FUNCTION_BLOCK T_Cylinder IMPLEMENTS I_Cylinder
VAR_INPUT
END_VAR
VAR_OUTPUT
END_VAR
VAR
	output AT %Q* : BOOL;
END_VAR

METHOD PUBLIC Extend
VAR_INPUT
END_VAR
output := true;
END_METHOD

METHOD PUBLIC Retract
VAR_INPUT
END_VAR
output := false;
END_METHOD

END_FUNCTION_BLOCK

(* stored: Version 1.1.0.1, ProductVersion 3.1.4024.4
   POU T_Cylinder: Id {c63bce25-1b52-4e4c-8ee8-d2fd9e9d433d}, SpecialFunc None
   Method Extend: Id {cf5fa276-c409-4304-ad6f-33b500cc5c85}
   Method Retract: Id {6bca65bb-c7e5-4db3-a695-e9b3a6428a17} *)
